// TIA Portal V19 export
TYPE "C402_VAR_VKL_TYPIC"
   STRUCT
      STS { ExternalAccessible := 'False'; ExternalVisible := 'False'; ExternalWritable := 'False'} : USInt;   // Actuele status van het verkeerslicht
      BMO { ExternalAccessible := 'False'; ExternalVisible := 'False'; ExternalWritable := 'False'} : USInt;   // Bedieningsmode
      BST { ExternalAccessible := 'False'; ExternalVisible := 'False'; ExternalWritable := 'False'} : USInt;   // Bestuurbaarheid
   END_STRUCT;
END_TYPE
